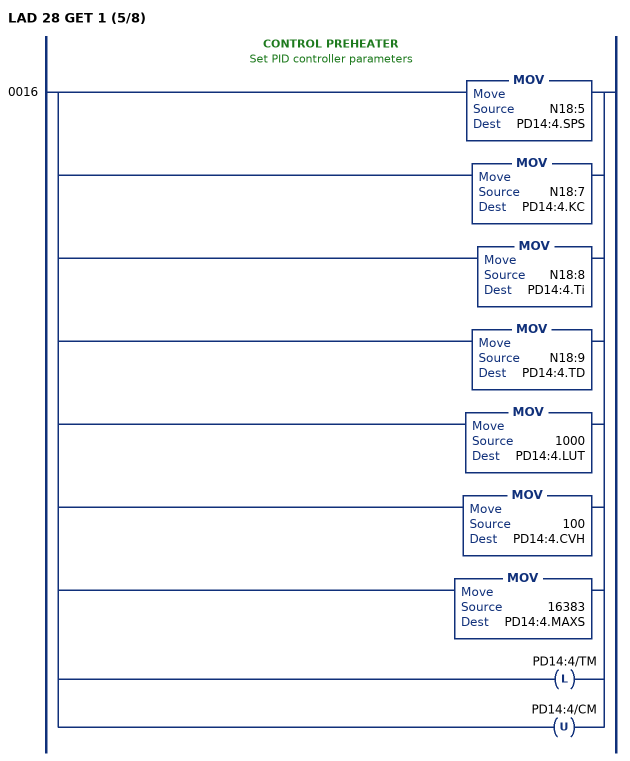
% Rung: 16 %
% TITLE: CONTROL PREHEATER %
% Set PID controller parameters %
SOR BST MOV N18:5 PD14:4.SPS NXB MOV N18:7 PD14:4.KC NXB MOV N18:8 PD14:4.Ti NXB MOV N18:9 PD14:4.TD NXB MOV 1000 PD14:4.LUT NXB MOV 100 PD14:4.CVH NXB MOV 16383 PD14:4.MAXS NXB OTL PD14:4/TM NXB OTU PD14:4/CM BND EOR
%   N18:5  GETTER_PH_SP  "<datalog>" %
%   N18:7  GET_PH_PID_GAIN %
%   N18:8  GET_PH_PID_INTEG %
%   N18:9  GET_PH_PID_DERIV %

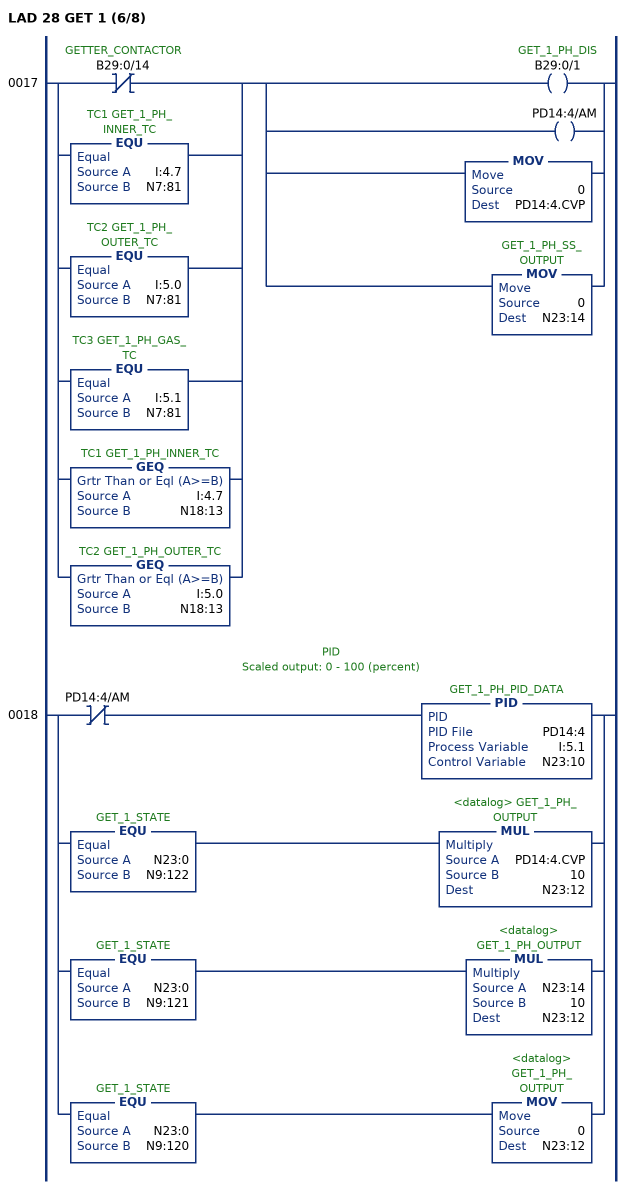
% Rung: 17 %
SOR BST XIO B29:0/14 NXB EQU I:4.7 N7:81 NXB EQU I:5.0 N7:81 NXB EQU I:5.1 N7:81 NXB GEQ I:4.7 N18:13 NXB GEQ I:5.0 N18:13 BND BST OTE B29:0/1 NXB OTE PD14:4/AM NXB MOV 0 PD14:4.CVP NXB MOV 0 N23:14 BND EOR
%   B29:0/14  GETTER_CONTACTOR %
%   I:4.7  GET_1_PH_INNER_TC  "TC1" %
%   N7:81  TC_OPEN_SP  "CONFIG The value read by an open TC input" %
%   I:5.0  GET_1_PH_OUTER_TC  "TC2" %
%   I:5.1  GET_1_PH_GAS_TC  "TC3" %
%   N18:13  GET_PH_ROD_LIMIT %
%   B29:0/1  GET_1_PH_DIS %
%   N23:14  GET_1_PH_SS_OUTPUT %
% Rung: 18 %
% PID
% Scaled output: 0 - 100 (percent) %
SOR BST XIO PD14:4/AM PID PD14:4 I:5.1 N23:10 NXB EQU N23:0 N9:122 MUL PD14:4.CVP 10 N23:12 NXB EQU N23:0 N9:121 MUL N23:14 10 N23:12 NXB EQU N23:0 N9:120 MOV 0 N23:12 BND EOR
%   PD14:4  GET_1_PH_PID_DATA %
%   I:5.1  GET_1_PH_GAS_TC  "TC3" %
%   N23:10  GET_1_PH_OUT_RAW %
%   N23:0  GET_1_STATE %
%   N9:122  GETTER_PURIFYING %
%   N23:12  GET_1_PH_OUTPUT  "<datalog>" %
%   N9:121  GETTER_SOFTSTART %
%   N23:14  GET_1_PH_SS_OUTPUT %
%   N9:120  GETTER_STANDBY %

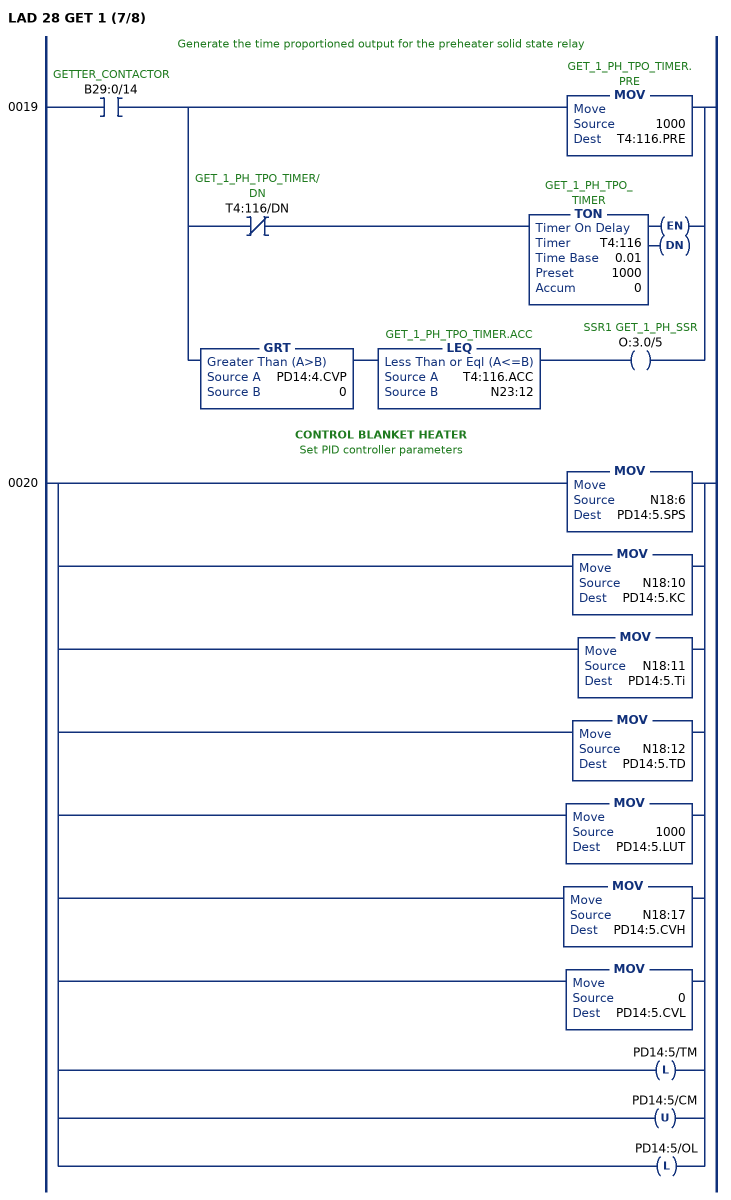
% Rung: 19 %
% Generate the time proportioned output for the preheater solid state relay %
SOR XIC B29:0/14 BST MOV 1000 T4:116.PRE NXB XIO T4:116/DN TON T4:116 0.01 1000 0 NXB GRT PD14:4.CVP 0 LEQ T4:116.ACC N23:12 OTE O:3.0/5 BND EOR
%   B29:0/14  GETTER_CONTACTOR %
%   T4:116  GET_1_PH_TPO_TIMER %
%   N23:12  GET_1_PH_OUTPUT  "<datalog>" %
%   O:3.0/5  GET_1_PH_SSR  "SSR1" %
% Rung: 20 %
% TITLE: CONTROL BLANKET HEATER %
% Set PID controller parameters %
SOR BST MOV N18:6 PD14:5.SPS NXB MOV N18:10 PD14:5.KC NXB MOV N18:11 PD14:5.Ti NXB MOV N18:12 PD14:5.TD NXB MOV 1000 PD14:5.LUT NXB MOV N18:17 PD14:5.CVH NXB MOV 0 PD14:5.CVL NXB OTL PD14:5/TM NXB OTU PD14:5/CM NXB OTL PD14:5/OL BND EOR
%   N18:6  GETTER_BLKT_SP  "<datalog>" %
%   N18:10  GET_BLKT_PID_GAIN %
%   N18:11  GET_BLKT_PID_INTEG %
%   N18:12  GET_BLKT_PID_DERIV %
%   N18:17  GET_BLKT_PID_HI_LIM %

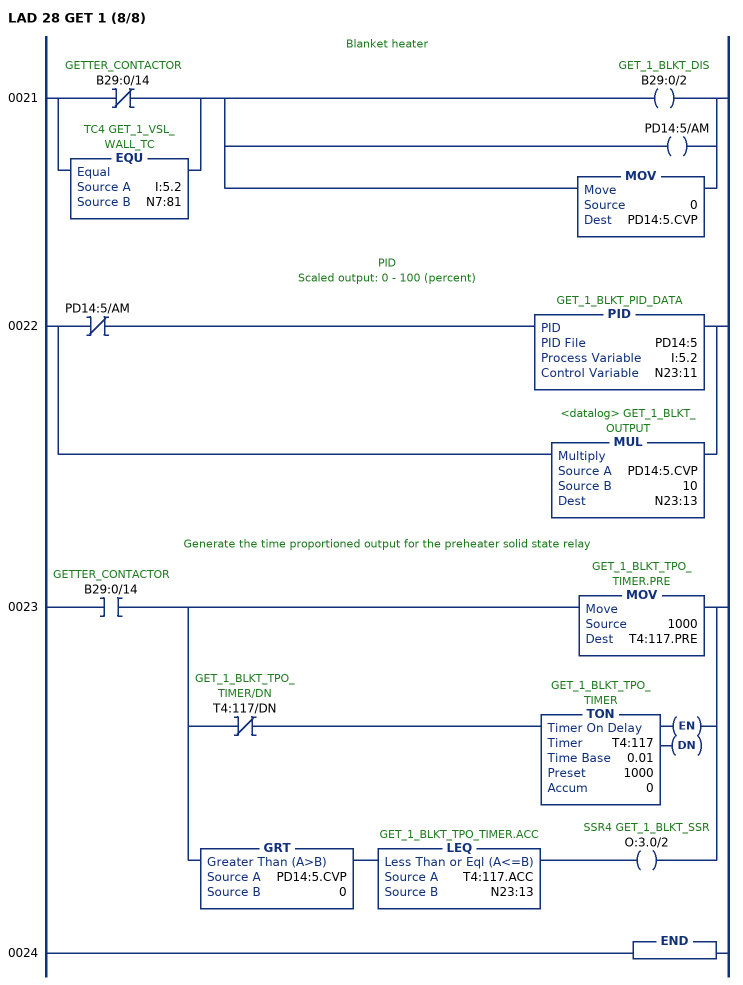
% Rung: 21 %
% Blanket heater %
SOR BST XIO B29:0/14 NXB EQU I:5.2 N7:81 BND BST OTE B29:0/2 NXB OTE PD14:5/AM NXB MOV 0 PD14:5.CVP BND EOR
%   B29:0/14  GETTER_CONTACTOR %
%   I:5.2  GET_1_VSL_WALL_TC  "TC4" %
%   N7:81  TC_OPEN_SP  "CONFIG The value read by an open TC input" %
%   B29:0/2  GET_1_BLKT_DIS %
% Rung: 22 %
% PID
% Scaled output: 0 - 100 (percent) %
SOR BST XIO PD14:5/AM PID PD14:5 I:5.2 N23:11 NXB MUL PD14:5.CVP 10 N23:13 BND EOR
%   PD14:5  GET_1_BLKT_PID_DATA %
%   I:5.2  GET_1_VSL_WALL_TC  "TC4" %
%   N23:11  GET_1_BLKT_OUT_RAW %
%   N23:13  GET_1_BLKT_OUTPUT  "<datalog>" %
% Rung: 23 %
% Generate the time proportioned output for the preheater solid state relay %
SOR XIC B29:0/14 BST MOV 1000 T4:117.PRE NXB XIO T4:117/DN TON T4:117 0.01 1000 0 NXB GRT PD14:5.CVP 0 LEQ T4:117.ACC N23:13 OTE O:3.0/2 BND EOR
%   B29:0/14  GETTER_CONTACTOR %
%   T4:117  GET_1_BLKT_TPO_TIMER %
%   N23:13  GET_1_BLKT_OUTPUT  "<datalog>" %
%   O:3.0/2  GET_1_BLKT_SSR  "SSR4" %
% Rung: 24 %
SOR END EOR

LADDER 29 "GET 2 FLT"
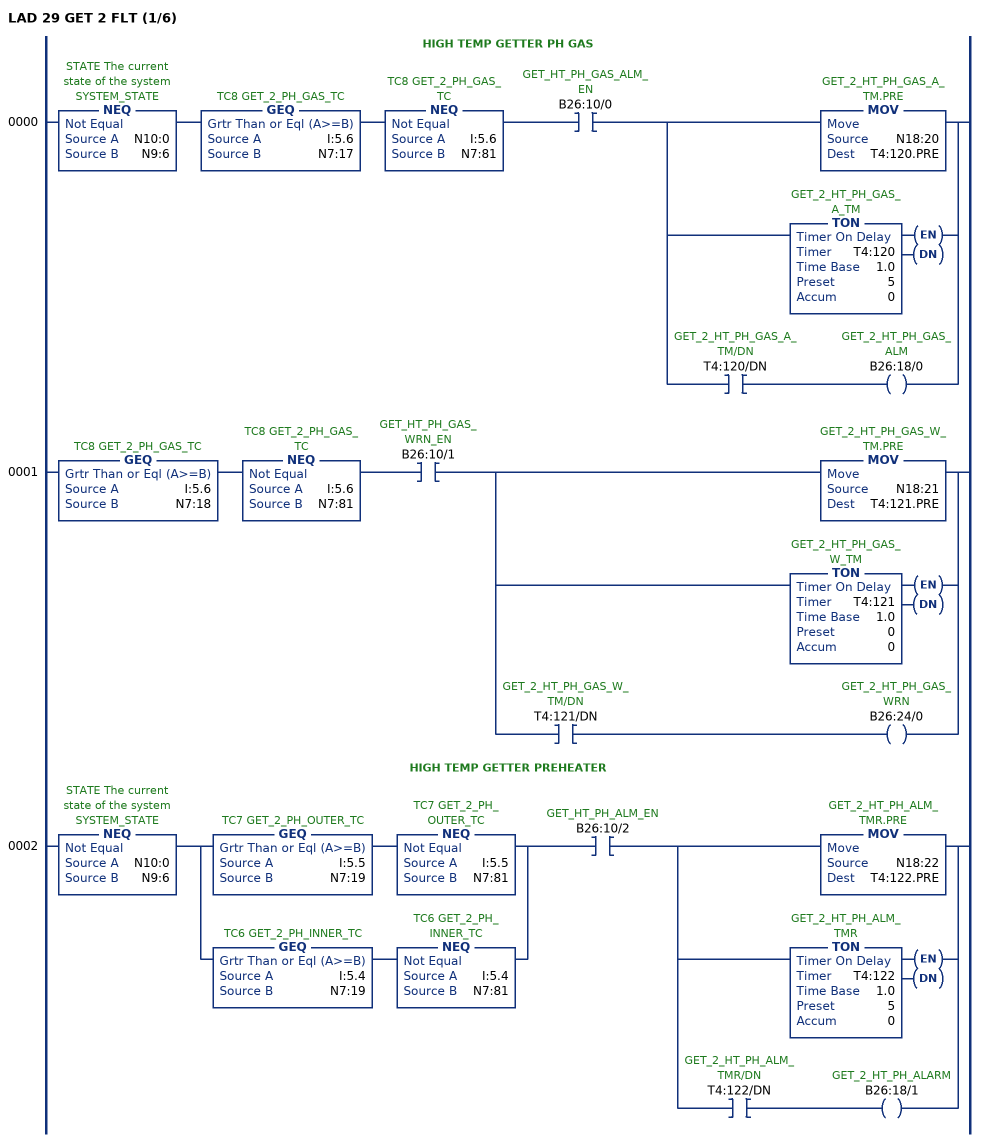
% Rung: 0 %
% TITLE: HIGH TEMP GETTER PH GAS %
SOR NEQ N10:0 N9:6 GEQ I:5.6 N7:17 NEQ I:5.6 N7:81 XIC B26:10/0 BST MOV N18:20 T4:120.PRE NXB TON T4:120 1.0 5 0 NXB XIC T4:120/DN OTE B26:18/0 BND EOR
%   N10:0  SYSTEM_STATE  "STATE The current state of the system" %
%   N9:6  SYSTEM_PURGE %
%   I:5.6  GET_2_PH_GAS_TC  "TC8" %
%   N7:17  GET_HT_PH_GAS_ALM_SP %
%   N7:81  TC_OPEN_SP  "CONFIG The value read by an open TC input" %
%   B26:10/0  GET_HT_PH_GAS_ALM_EN %
%   N18:20  GET_HT_PH_GAS_ALM_DL %
%   T4:120  GET_2_HT_PH_GAS_A_TM %
%   B26:18/0  GET_2_HT_PH_GAS_ALM %
% Rung: 1 %
SOR GEQ I:5.6 N7:18 NEQ I:5.6 N7:81 XIC B26:10/1 BST MOV N18:21 T4:121.PRE NXB TON T4:121 1.0 0 0 NXB XIC T4:121/DN OTE B26:24/0 BND EOR
%   I:5.6  GET_2_PH_GAS_TC  "TC8" %
%   N7:18  GET_HT_PH_GAS_WRN_SP %
%   N7:81  TC_OPEN_SP  "CONFIG The value read by an open TC input" %
%   B26:10/1  GET_HT_PH_GAS_WRN_EN %
%   N18:21  GET_HT_PH_GAS_WRN_DL %
%   T4:121  GET_2_HT_PH_GAS_W_TM %
%   B26:24/0  GET_2_HT_PH_GAS_WRN %
% Rung: 2 %
% TITLE: HIGH TEMP GETTER PREHEATER %
SOR NEQ N10:0 N9:6 BST GEQ I:5.5 N7:19 NEQ I:5.5 N7:81 NXB GEQ I:5.4 N7:19 NEQ I:5.4 N7:81 BND XIC B26:10/2 BST MOV N18:22 T4:122.PRE NXB TON T4:122 1.0 5 0 NXB XIC T4:122/DN OTE B26:18/1 BND EOR
%   N10:0  SYSTEM_STATE  "STATE The current state of the system" %
%   N9:6  SYSTEM_PURGE %
%   I:5.5  GET_2_PH_OUTER_TC  "TC7" %
%   N7:19  GET_HT_PH_ALM_SP %
%   N7:81  TC_OPEN_SP  "CONFIG The value read by an open TC input" %
%   I:5.4  GET_2_PH_INNER_TC  "TC6" %
%   B26:10/2  GET_HT_PH_ALM_EN %
%   N18:22  GET_HT_PH_ALM_DLY %
%   T4:122  GET_2_HT_PH_ALM_TMR %
%   B26:18/1  GET_2_HT_PH_ALARM %

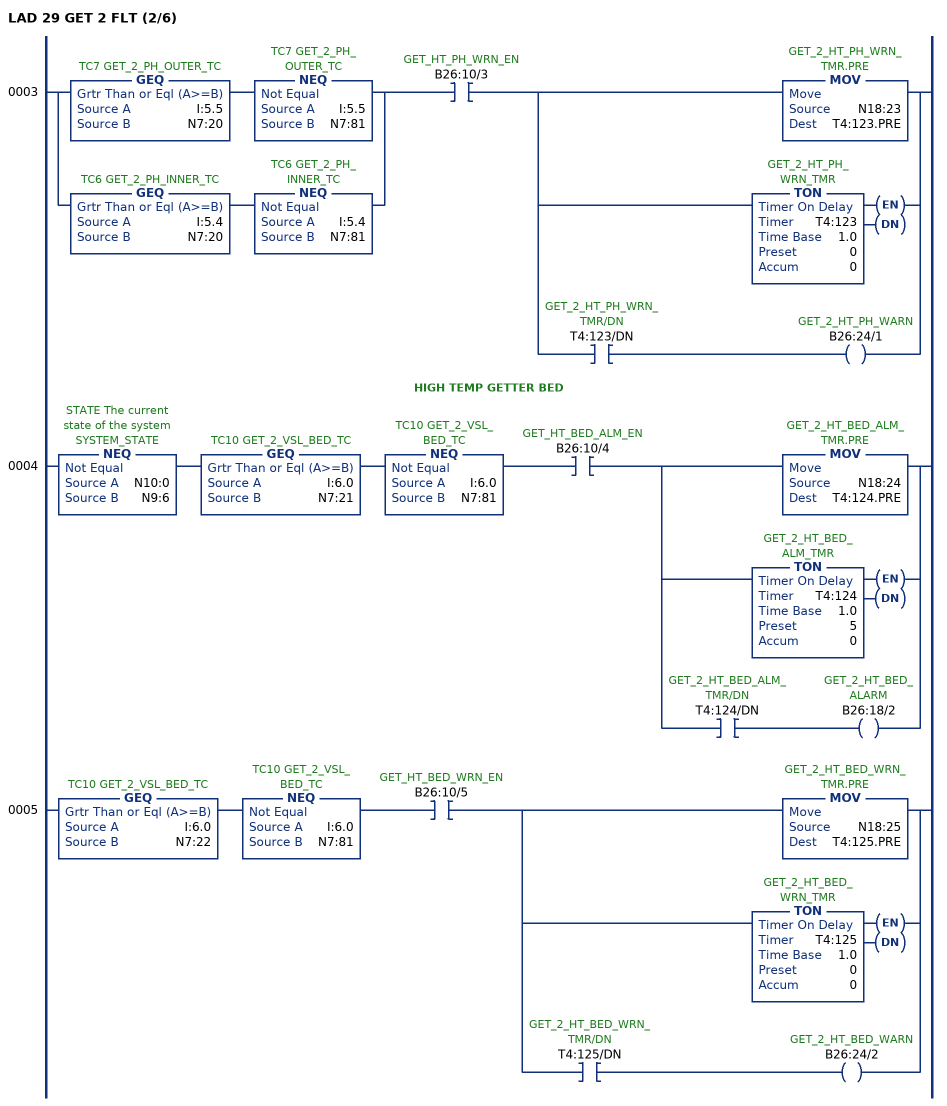
% Rung: 3 %
SOR BST GEQ I:5.5 N7:20 NEQ I:5.5 N7:81 NXB GEQ I:5.4 N7:20 NEQ I:5.4 N7:81 BND XIC B26:10/3 BST MOV N18:23 T4:123.PRE NXB TON T4:123 1.0 0 0 NXB XIC T4:123/DN OTE B26:24/1 BND EOR
%   I:5.5  GET_2_PH_OUTER_TC  "TC7" %
%   N7:20  GET_HT_PH_WRN_SP %
%   N7:81  TC_OPEN_SP  "CONFIG The value read by an open TC input" %
%   I:5.4  GET_2_PH_INNER_TC  "TC6" %
%   B26:10/3  GET_HT_PH_WRN_EN %
%   N18:23  GET_HT_PH_WRN_DLY %
%   T4:123  GET_2_HT_PH_WRN_TMR %
%   B26:24/1  GET_2_HT_PH_WARN %
% Rung: 4 %
% TITLE: HIGH TEMP GETTER BED %
SOR NEQ N10:0 N9:6 GEQ I:6.0 N7:21 NEQ I:6.0 N7:81 XIC B26:10/4 BST MOV N18:24 T4:124.PRE NXB TON T4:124 1.0 5 0 NXB XIC T4:124/DN OTE B26:18/2 BND EOR
%   N10:0  SYSTEM_STATE  "STATE The current state of the system" %
%   N9:6  SYSTEM_PURGE %
%   I:6.0  GET_2_VSL_BED_TC  "TC10" %
%   N7:21  GET_HT_BED_ALM_SP %
%   N7:81  TC_OPEN_SP  "CONFIG The value read by an open TC input" %
%   B26:10/4  GET_HT_BED_ALM_EN %
%   N18:24  GET_HT_BED_ALM_DLY %
%   T4:124  GET_2_HT_BED_ALM_TMR %
%   B26:18/2  GET_2_HT_BED_ALARM %
% Rung: 5 %
SOR GEQ I:6.0 N7:22 NEQ I:6.0 N7:81 XIC B26:10/5 BST MOV N18:25 T4:125.PRE NXB TON T4:125 1.0 0 0 NXB XIC T4:125/DN OTE B26:24/2 BND EOR
%   I:6.0  GET_2_VSL_BED_TC  "TC10" %
%   N7:22  GET_HT_BED_WRN_SP %
%   N7:81  TC_OPEN_SP  "CONFIG The value read by an open TC input" %
%   B26:10/5  GET_HT_BED_WRN_EN %
%   N18:25  GET_HT_BED_WRN_DLY %
%   T4:125  GET_2_HT_BED_WRN_TMR %
%   B26:24/2  GET_2_HT_BED_WARN %

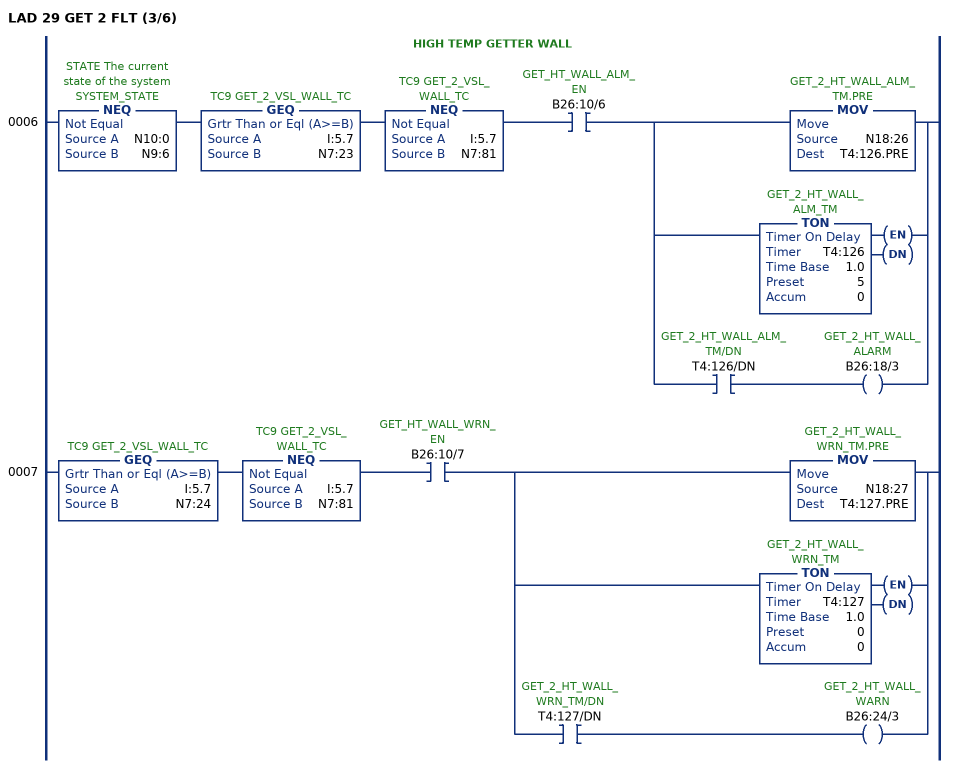
% Rung: 6 %
% TITLE: HIGH TEMP GETTER WALL %
SOR NEQ N10:0 N9:6 GEQ I:5.7 N7:23 NEQ I:5.7 N7:81 XIC B26:10/6 BST MOV N18:26 T4:126.PRE NXB TON T4:126 1.0 5 0 NXB XIC T4:126/DN OTE B26:18/3 BND EOR
%   N10:0  SYSTEM_STATE  "STATE The current state of the system" %
%   N9:6  SYSTEM_PURGE %
%   I:5.7  GET_2_VSL_WALL_TC  "TC9" %
%   N7:23  GET_HT_WALL_ALM_SP %
%   N7:81  TC_OPEN_SP  "CONFIG The value read by an open TC input" %
%   B26:10/6  GET_HT_WALL_ALM_EN %
%   N18:26  GET_HT_WALL_ALM_DLY %
%   T4:126  GET_2_HT_WALL_ALM_TM %
%   B26:18/3  GET_2_HT_WALL_ALARM %
% Rung: 7 %
SOR GEQ I:5.7 N7:24 NEQ I:5.7 N7:81 XIC B26:10/7 BST MOV N18:27 T4:127.PRE NXB TON T4:127 1.0 0 0 NXB XIC T4:127/DN OTE B26:24/3 BND EOR
%   I:5.7  GET_2_VSL_WALL_TC  "TC9" %
%   N7:24  GET_HT_WALL_WRN_SP %
%   N7:81  TC_OPEN_SP  "CONFIG The value read by an open TC input" %
%   B26:10/7  GET_HT_WALL_WRN_EN %
%   N18:27  GET_HT_WALL_WRN_DLY %
%   T4:127  GET_2_HT_WALL_WRN_TM %
%   B26:24/3  GET_2_HT_WALL_WARN %

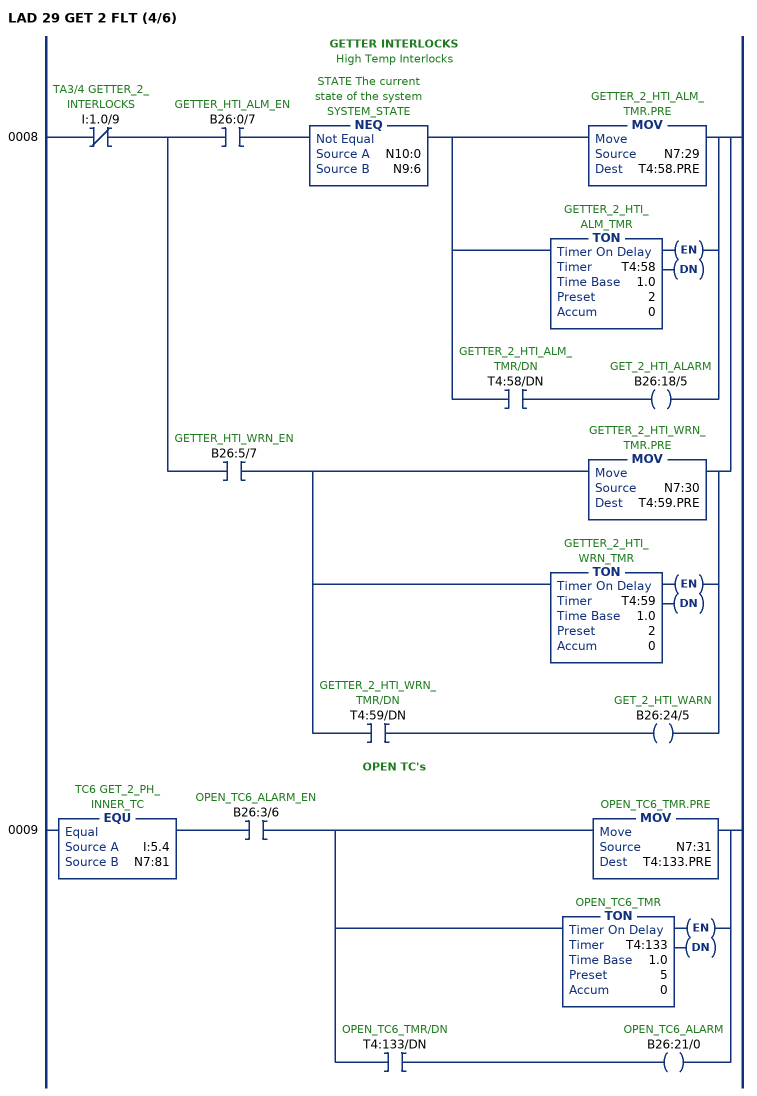
% Rung: 8 %
% TITLE: GETTER INTERLOCKS %
% High Temp Interlocks %
SOR XIO I:1.0/9 BST XIC B26:0/7 NEQ N10:0 N9:6 BST MOV N7:29 T4:58.PRE NXB TON T4:58 1.0 2 0 NXB XIC T4:58/DN OTE B26:18/5 BND NXB XIC B26:5/7 BST MOV N7:30 T4:59.PRE NXB TON T4:59 1.0 2 0 NXB XIC T4:59/DN OTE B26:24/5 BND BND EOR
%   I:1.0/9  GETTER_2_INTERLOCKS  "TA3/4" %
%   B26:0/7  GETTER_HTI_ALM_EN %
%   N10:0  SYSTEM_STATE  "STATE The current state of the system" %
%   N9:6  SYSTEM_PURGE %
%   N7:29  GETTER_HTI_ALM_DLY %
%   T4:58  GETTER_2_HTI_ALM_TMR %
%   B26:18/5  GET_2_HTI_ALARM %
%   B26:5/7  GETTER_HTI_WRN_EN %
%   N7:30  GETTER_HTI_WRN_DLY %
%   T4:59  GETTER_2_HTI_WRN_TMR %
%   B26:24/5  GET_2_HTI_WARN %
% Rung: 9 %
% TITLE: OPEN TC's %
SOR EQU I:5.4 N7:81 XIC B26:3/6 BST MOV N7:31 T4:133.PRE NXB TON T4:133 1.0 5 0 NXB XIC T4:133/DN OTE B26:21/0 BND EOR
%   I:5.4  GET_2_PH_INNER_TC  "TC6" %
%   N7:81  TC_OPEN_SP  "CONFIG The value read by an open TC input" %
%   B26:3/6  OPEN_TC6_ALARM_EN %
%   N7:31  OPEN_TC_DLY %
%   T4:133  OPEN_TC6_TMR %
%   B26:21/0  OPEN_TC6_ALARM %

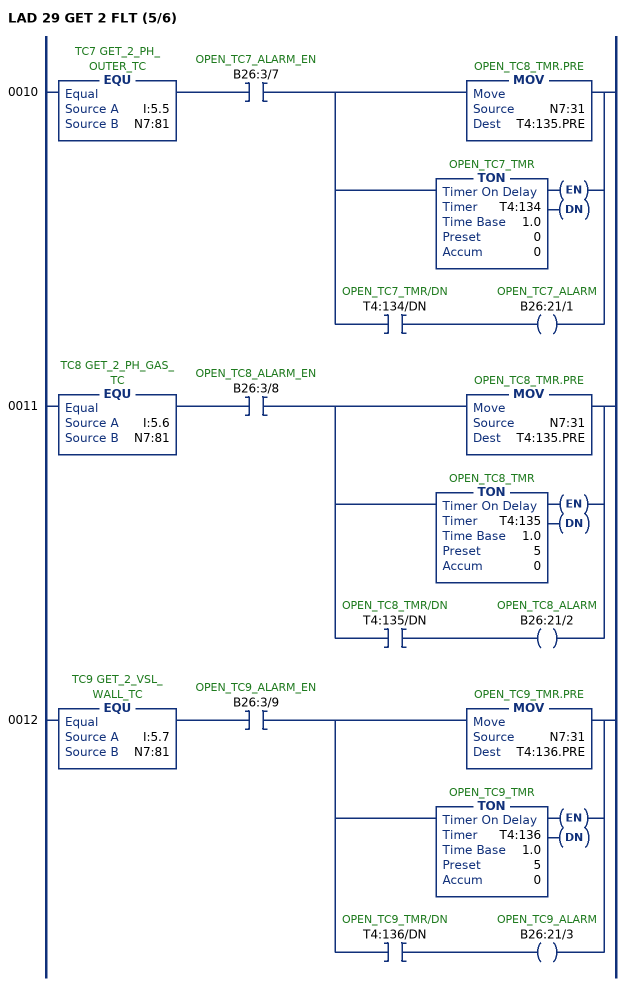
% Rung: 10 %
SOR EQU I:5.5 N7:81 XIC B26:3/7 BST MOV N7:31 T4:135.PRE NXB TON T4:134 1.0 0 0 NXB XIC T4:134/DN OTE B26:21/1 BND EOR
%   I:5.5  GET_2_PH_OUTER_TC  "TC7" %
%   N7:81  TC_OPEN_SP  "CONFIG The value read by an open TC input" %
%   B26:3/7  OPEN_TC7_ALARM_EN %
%   N7:31  OPEN_TC_DLY %
%   T4:135  OPEN_TC8_TMR %
%   T4:134  OPEN_TC7_TMR %
%   B26:21/1  OPEN_TC7_ALARM %
% Rung: 11 %
SOR EQU I:5.6 N7:81 XIC B26:3/8 BST MOV N7:31 T4:135.PRE NXB TON T4:135 1.0 5 0 NXB XIC T4:135/DN OTE B26:21/2 BND EOR
%   I:5.6  GET_2_PH_GAS_TC  "TC8" %
%   N7:81  TC_OPEN_SP  "CONFIG The value read by an open TC input" %
%   B26:3/8  OPEN_TC8_ALARM_EN %
%   N7:31  OPEN_TC_DLY %
%   T4:135  OPEN_TC8_TMR %
%   B26:21/2  OPEN_TC8_ALARM %
% Rung: 12 %
SOR EQU I:5.7 N7:81 XIC B26:3/9 BST MOV N7:31 T4:136.PRE NXB TON T4:136 1.0 5 0 NXB XIC T4:136/DN OTE B26:21/3 BND EOR
%   I:5.7  GET_2_VSL_WALL_TC  "TC9" %
%   N7:81  TC_OPEN_SP  "CONFIG The value read by an open TC input" %
%   B26:3/9  OPEN_TC9_ALARM_EN %
%   N7:31  OPEN_TC_DLY %
%   T4:136  OPEN_TC9_TMR %
%   B26:21/3  OPEN_TC9_ALARM %

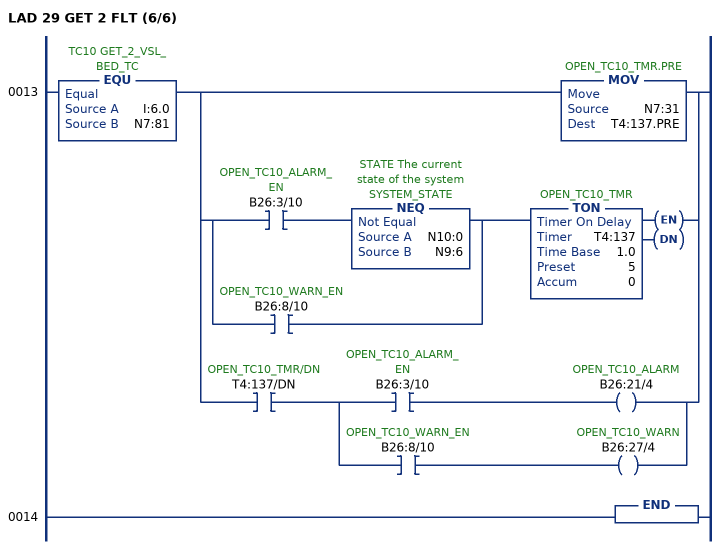
% Rung: 13 %
SOR EQU I:6.0 N7:81 BST MOV N7:31 T4:137.PRE NXB BST XIC B26:3/10 NEQ N10:0 N9:6 NXB XIC B26:8/10 BND TON T4:137 1.0 5 0 NXB XIC T4:137/DN BST XIC B26:3/10 OTE B26:21/4 NXB XIC B26:8/10 OTE B26:27/4 BND BND EOR
%   I:6.0  GET_2_VSL_BED_TC  "TC10" %
%   N7:81  TC_OPEN_SP  "CONFIG The value read by an open TC input" %
%   N7:31  OPEN_TC_DLY %
%   T4:137  OPEN_TC10_TMR %
%   B26:3/10  OPEN_TC10_ALARM_EN %
%   N10:0  SYSTEM_STATE  "STATE The current state of the system" %
%   N9:6  SYSTEM_PURGE %
%   B26:8/10  OPEN_TC10_WARN_EN %
%   B26:21/4  OPEN_TC10_ALARM %
%   B26:27/4  OPEN_TC10_WARN %
% Rung: 14 %
SOR END EOR

LADDER 30 "GET 2"
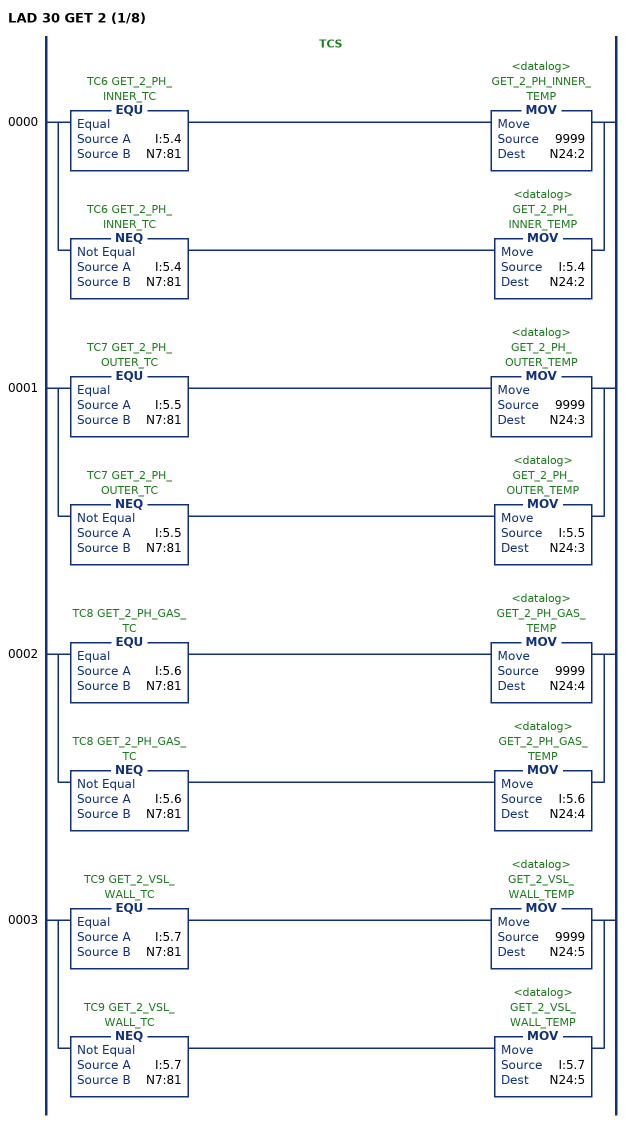
% Rung: 0 %
% TITLE: TCS %
SOR BST EQU I:5.4 N7:81 MOV 9999 N24:2 NXB NEQ I:5.4 N7:81 MOV I:5.4 N24:2 BND EOR
%   I:5.4  GET_2_PH_INNER_TC  "TC6" %
%   N7:81  TC_OPEN_SP  "CONFIG The value read by an open TC input" %
%   N24:2  GET_2_PH_INNER_TEMP  "<datalog>" %
% Rung: 1 %
SOR BST EQU I:5.5 N7:81 MOV 9999 N24:3 NXB NEQ I:5.5 N7:81 MOV I:5.5 N24:3 BND EOR
%   I:5.5  GET_2_PH_OUTER_TC  "TC7" %
%   N7:81  TC_OPEN_SP  "CONFIG The value read by an open TC input" %
%   N24:3  GET_2_PH_OUTER_TEMP  "<datalog>" %
% Rung: 2 %
SOR BST EQU I:5.6 N7:81 MOV 9999 N24:4 NXB NEQ I:5.6 N7:81 MOV I:5.6 N24:4 BND EOR
%   I:5.6  GET_2_PH_GAS_TC  "TC8" %
%   N7:81  TC_OPEN_SP  "CONFIG The value read by an open TC input" %
%   N24:4  GET_2_PH_GAS_TEMP  "<datalog>" %
% Rung: 3 %
SOR BST EQU I:5.7 N7:81 MOV 9999 N24:5 NXB NEQ I:5.7 N7:81 MOV I:5.7 N24:5 BND EOR
%   I:5.7  GET_2_VSL_WALL_TC  "TC9" %
%   N7:81  TC_OPEN_SP  "CONFIG The value read by an open TC input" %
%   N24:5  GET_2_VSL_WALL_TEMP  "<datalog>" %

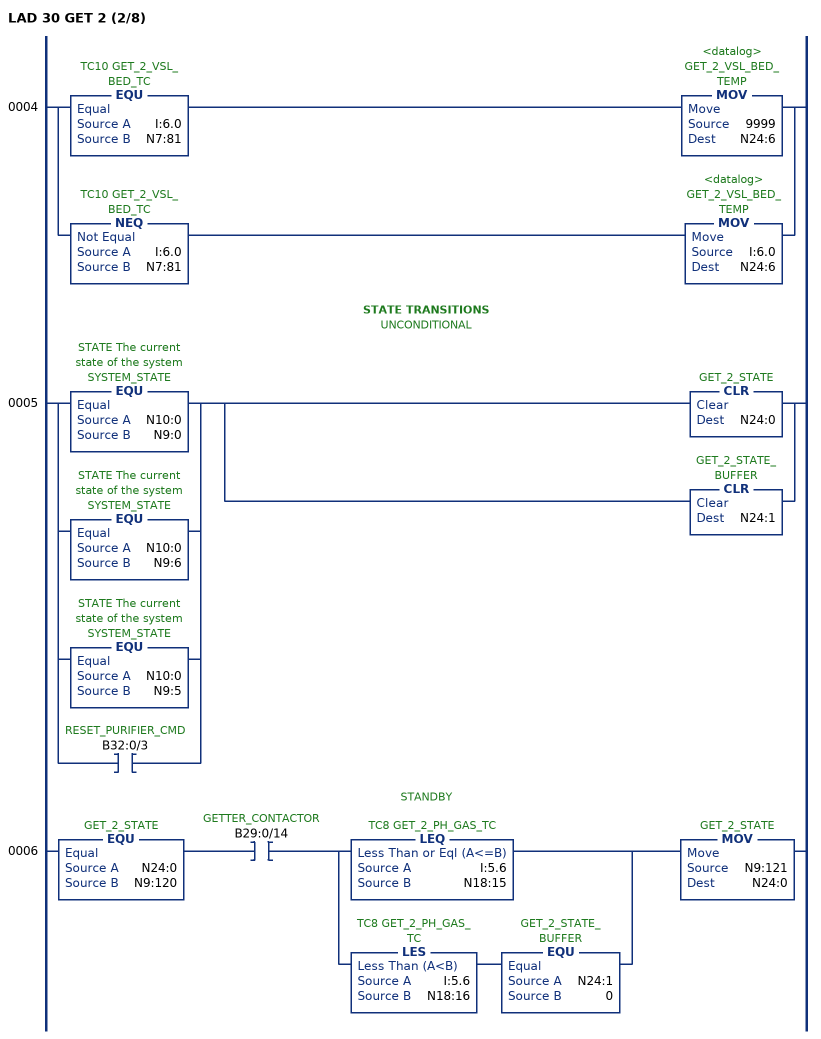
% Rung: 4 %
SOR BST EQU I:6.0 N7:81 MOV 9999 N24:6 NXB NEQ I:6.0 N7:81 MOV I:6.0 N24:6 BND EOR
%   I:6.0  GET_2_VSL_BED_TC  "TC10" %
%   N7:81  TC_OPEN_SP  "CONFIG The value read by an open TC input" %
%   N24:6  GET_2_VSL_BED_TEMP  "<datalog>" %
% Rung: 5 %
% TITLE: STATE TRANSITIONS %
% UNCONDITIONAL %
SOR BST EQU N10:0 N9:0 NXB EQU N10:0 N9:6 NXB EQU N10:0 N9:5 NXB XIC B32:0/3 BND BST CLR N24:0 NXB CLR N24:1 BND EOR
%   N10:0  SYSTEM_STATE  "STATE The current state of the system" %
%   N9:0  SYSTEM_OFFLINE %
%   N9:6  SYSTEM_PURGE %
%   N9:5  SYSTEM_QUICK_START %
%   B32:0/3  RESET_PURIFIER_CMD %
%   N24:0  GET_2_STATE %
%   N24:1  GET_2_STATE_BUFFER %
% Rung: 6 %
% STANDBY %
SOR EQU N24:0 N9:120 XIC B29:0/14 BST LEQ I:5.6 N18:15 NXB LES I:5.6 N18:16 EQU N24:1 0 BND MOV N9:121 N24:0 EOR
%   N24:0  GET_2_STATE %
%   N9:120  GETTER_STANDBY %
%   B29:0/14  GETTER_CONTACTOR %
%   I:5.6  GET_2_PH_GAS_TC  "TC8" %
%   N18:15  GETTER_SS_BEGIN_TEMP %
%   N18:16  GETTER_SS_END_TEMP %
%   N24:1  GET_2_STATE_BUFFER %
%   N9:121  GETTER_SOFTSTART %

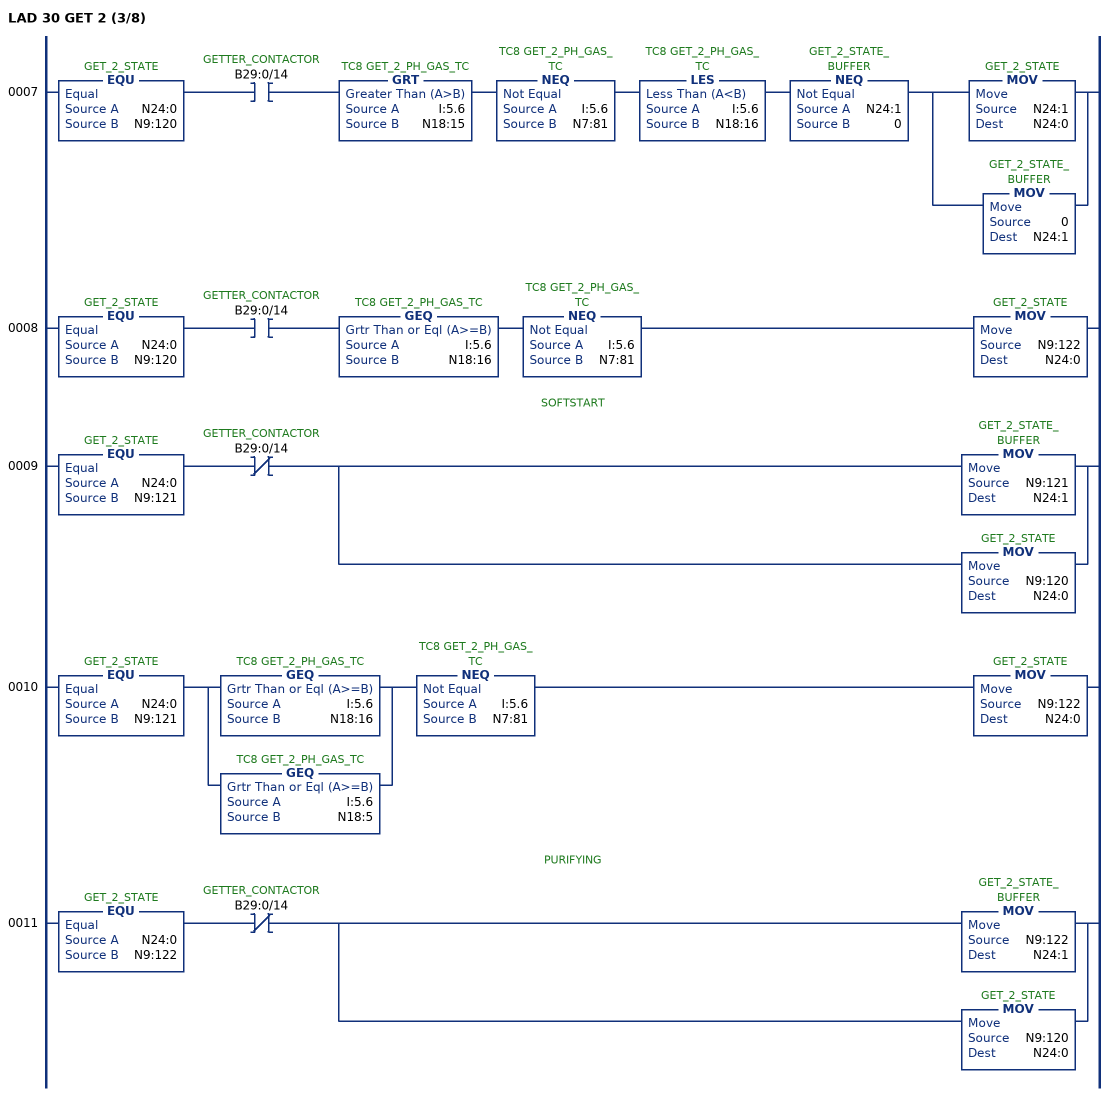
% Rung: 7 %
SOR EQU N24:0 N9:120 XIC B29:0/14 GRT I:5.6 N18:15 NEQ I:5.6 N7:81 LES I:5.6 N18:16 NEQ N24:1 0 BST MOV N24:1 N24:0 NXB MOV 0 N24:1 BND EOR
%   N24:0  GET_2_STATE %
%   N9:120  GETTER_STANDBY %
%   B29:0/14  GETTER_CONTACTOR %
%   I:5.6  GET_2_PH_GAS_TC  "TC8" %
%   N18:15  GETTER_SS_BEGIN_TEMP %
%   N7:81  TC_OPEN_SP  "CONFIG The value read by an open TC input" %
%   N18:16  GETTER_SS_END_TEMP %
%   N24:1  GET_2_STATE_BUFFER %
% Rung: 8 %
SOR EQU N24:0 N9:120 XIC B29:0/14 GEQ I:5.6 N18:16 NEQ I:5.6 N7:81 MOV N9:122 N24:0 EOR
%   N24:0  GET_2_STATE %
%   N9:120  GETTER_STANDBY %
%   B29:0/14  GETTER_CONTACTOR %
%   I:5.6  GET_2_PH_GAS_TC  "TC8" %
%   N18:16  GETTER_SS_END_TEMP %
%   N7:81  TC_OPEN_SP  "CONFIG The value read by an open TC input" %
%   N9:122  GETTER_PURIFYING %
% Rung: 9 %
% SOFTSTART %
SOR EQU N24:0 N9:121 XIO B29:0/14 BST MOV N9:121 N24:1 NXB MOV N9:120 N24:0 BND EOR
%   N24:0  GET_2_STATE %
%   N9:121  GETTER_SOFTSTART %
%   B29:0/14  GETTER_CONTACTOR %
%   N24:1  GET_2_STATE_BUFFER %
%   N9:120  GETTER_STANDBY %
% Rung: 10 %
SOR EQU N24:0 N9:121 BST GEQ I:5.6 N18:16 NXB GEQ I:5.6 N18:5 BND NEQ I:5.6 N7:81 MOV N9:122 N24:0 EOR
%   N24:0  GET_2_STATE %
%   N9:121  GETTER_SOFTSTART %
%   I:5.6  GET_2_PH_GAS_TC  "TC8" %
%   N18:16  GETTER_SS_END_TEMP %
%   N18:5  GETTER_PH_SP  "<datalog>" %
%   N7:81  TC_OPEN_SP  "CONFIG The value read by an open TC input" %
%   N9:122  GETTER_PURIFYING %
% Rung: 11 %
% PURIFYING %
SOR EQU N24:0 N9:122 XIO B29:0/14 BST MOV N9:122 N24:1 NXB MOV N9:120 N24:0 BND EOR
%   N24:0  GET_2_STATE %
%   N9:122  GETTER_PURIFYING %
%   B29:0/14  GETTER_CONTACTOR %
%   N24:1  GET_2_STATE_BUFFER %
%   N9:120  GETTER_STANDBY %

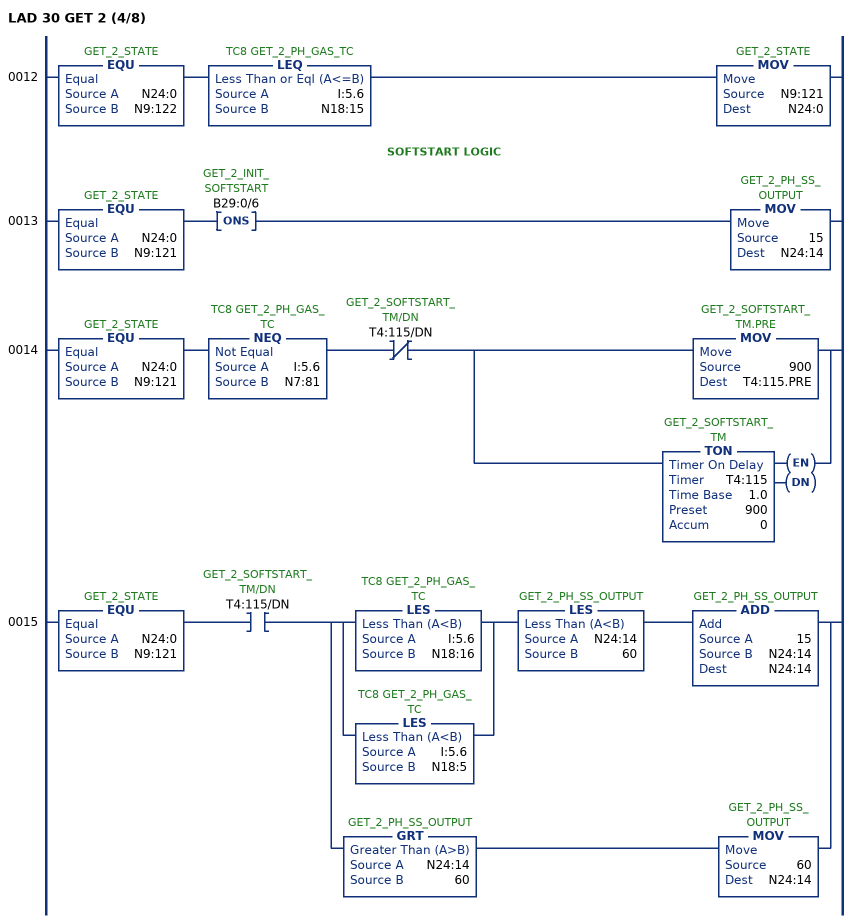
% Rung: 12 %
SOR EQU N24:0 N9:122 LEQ I:5.6 N18:15 MOV N9:121 N24:0 EOR
%   N24:0  GET_2_STATE %
%   N9:122  GETTER_PURIFYING %
%   I:5.6  GET_2_PH_GAS_TC  "TC8" %
%   N18:15  GETTER_SS_BEGIN_TEMP %
%   N9:121  GETTER_SOFTSTART %
% Rung: 13 %
% TITLE: SOFTSTART LOGIC %
SOR EQU N24:0 N9:121 ONS B29:0/6 MOV 15 N24:14 EOR
%   N24:0  GET_2_STATE %
%   N9:121  GETTER_SOFTSTART %
%   B29:0/6  GET_2_INIT_SOFTSTART %
%   N24:14  GET_2_PH_SS_OUTPUT %
% Rung: 14 %
SOR EQU N24:0 N9:121 NEQ I:5.6 N7:81 XIO T4:115/DN BST MOV 900 T4:115.PRE NXB TON T4:115 1.0 900 0 BND EOR
%   N24:0  GET_2_STATE %
%   N9:121  GETTER_SOFTSTART %
%   I:5.6  GET_2_PH_GAS_TC  "TC8" %
%   N7:81  TC_OPEN_SP  "CONFIG The value read by an open TC input" %
%   T4:115  GET_2_SOFTSTART_TM %
% Rung: 15 %
SOR EQU N24:0 N9:121 XIC T4:115/DN BST BST LES I:5.6 N18:16 NXB LES I:5.6 N18:5 BND LES N24:14 60 ADD 15 N24:14 N24:14 NXB GRT N24:14 60 MOV 60 N24:14 BND EOR
%   N24:0  GET_2_STATE %
%   N9:121  GETTER_SOFTSTART %
%   T4:115  GET_2_SOFTSTART_TM %
%   I:5.6  GET_2_PH_GAS_TC  "TC8" %
%   N18:16  GETTER_SS_END_TEMP %
%   N18:5  GETTER_PH_SP  "<datalog>" %
%   N24:14  GET_2_PH_SS_OUTPUT %

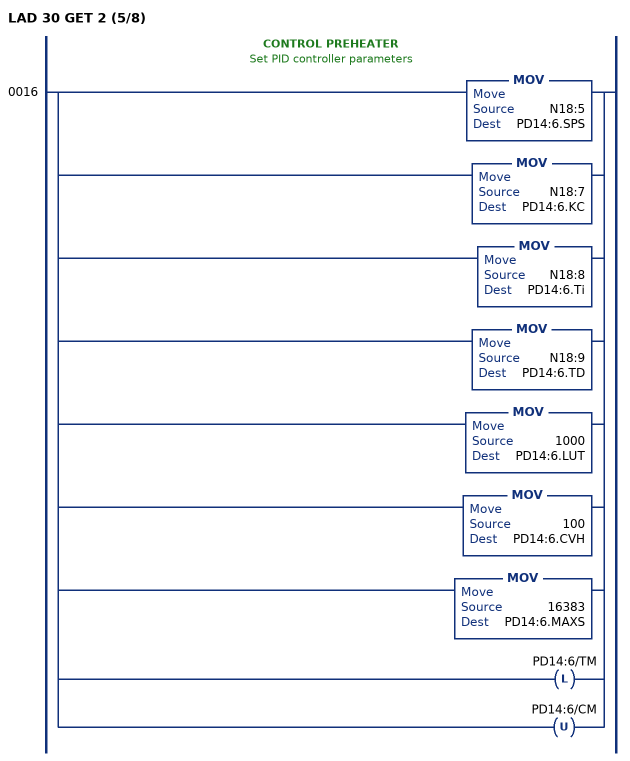
% Rung: 16 %
% TITLE: CONTROL PREHEATER %
% Set PID controller parameters %
SOR BST MOV N18:5 PD14:6.SPS NXB MOV N18:7 PD14:6.KC NXB MOV N18:8 PD14:6.Ti NXB MOV N18:9 PD14:6.TD NXB MOV 1000 PD14:6.LUT NXB MOV 100 PD14:6.CVH NXB MOV 16383 PD14:6.MAXS NXB OTL PD14:6/TM NXB OTU PD14:6/CM BND EOR
%   N18:5  GETTER_PH_SP  "<datalog>" %
%   N18:7  GET_PH_PID_GAIN %
%   N18:8  GET_PH_PID_INTEG %
%   N18:9  GET_PH_PID_DERIV %

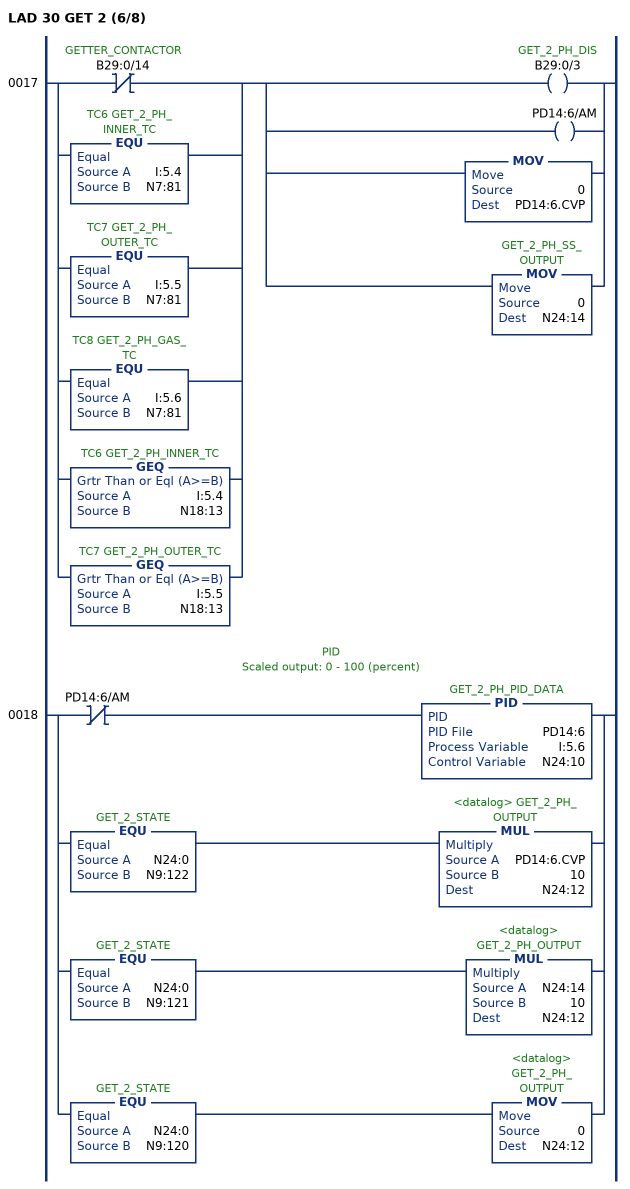
% Rung: 17 %
SOR BST XIO B29:0/14 NXB EQU I:5.4 N7:81 NXB EQU I:5.5 N7:81 NXB EQU I:5.6 N7:81 NXB GEQ I:5.4 N18:13 NXB GEQ I:5.5 N18:13 BND BST OTE B29:0/3 NXB OTE PD14:6/AM NXB MOV 0 PD14:6.CVP NXB MOV 0 N24:14 BND EOR
%   B29:0/14  GETTER_CONTACTOR %
%   I:5.4  GET_2_PH_INNER_TC  "TC6" %
%   N7:81  TC_OPEN_SP  "CONFIG The value read by an open TC input" %
%   I:5.5  GET_2_PH_OUTER_TC  "TC7" %
%   I:5.6  GET_2_PH_GAS_TC  "TC8" %
%   N18:13  GET_PH_ROD_LIMIT %
%   B29:0/3  GET_2_PH_DIS %
%   N24:14  GET_2_PH_SS_OUTPUT %
% Rung: 18 %
% PID
% Scaled output: 0 - 100 (percent) %
SOR BST XIO PD14:6/AM PID PD14:6 I:5.6 N24:10 NXB EQU N24:0 N9:122 MUL PD14:6.CVP 10 N24:12 NXB EQU N24:0 N9:121 MUL N24:14 10 N24:12 NXB EQU N24:0 N9:120 MOV 0 N24:12 BND EOR
%   PD14:6  GET_2_PH_PID_DATA %
%   I:5.6  GET_2_PH_GAS_TC  "TC8" %
%   N24:10  GET_2_PH_OUT_RAW %
%   N24:0  GET_2_STATE %
%   N9:122  GETTER_PURIFYING %
%   N24:12  GET_2_PH_OUTPUT  "<datalog>" %
%   N9:121  GETTER_SOFTSTART %
%   N24:14  GET_2_PH_SS_OUTPUT %
%   N9:120  GETTER_STANDBY %

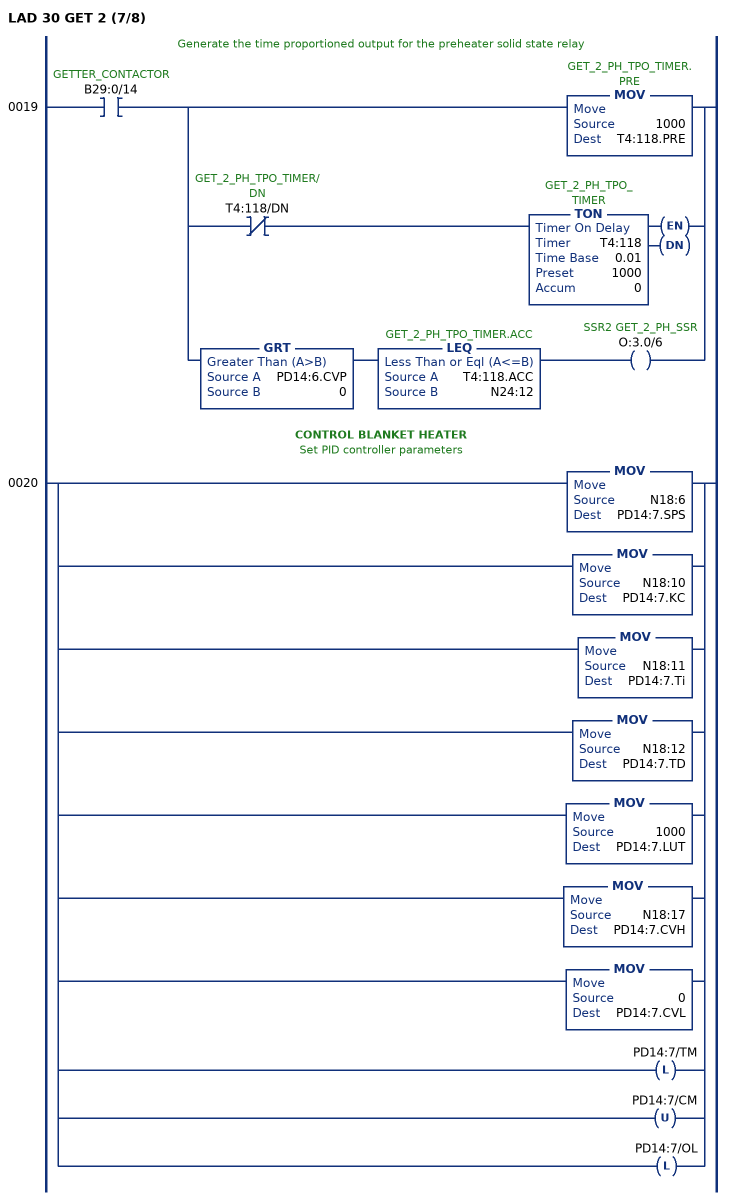
% Rung: 19 %
% Generate the time proportioned output for the preheater solid state relay %
SOR XIC B29:0/14 BST MOV 1000 T4:118.PRE NXB XIO T4:118/DN TON T4:118 0.01 1000 0 NXB GRT PD14:6.CVP 0 LEQ T4:118.ACC N24:12 OTE O:3.0/6 BND EOR
%   B29:0/14  GETTER_CONTACTOR %
%   T4:118  GET_2_PH_TPO_TIMER %
%   N24:12  GET_2_PH_OUTPUT  "<datalog>" %
%   O:3.0/6  GET_2_PH_SSR  "SSR2" %
% Rung: 20 %
% TITLE: CONTROL BLANKET HEATER %
% Set PID controller parameters %
SOR BST MOV N18:6 PD14:7.SPS NXB MOV N18:10 PD14:7.KC NXB MOV N18:11 PD14:7.Ti NXB MOV N18:12 PD14:7.TD NXB MOV 1000 PD14:7.LUT NXB MOV N18:17 PD14:7.CVH NXB MOV 0 PD14:7.CVL NXB OTL PD14:7/TM NXB OTU PD14:7/CM NXB OTL PD14:7/OL BND EOR
%   N18:6  GETTER_BLKT_SP  "<datalog>" %
%   N18:10  GET_BLKT_PID_GAIN %
%   N18:11  GET_BLKT_PID_INTEG %
%   N18:12  GET_BLKT_PID_DERIV %
%   N18:17  GET_BLKT_PID_HI_LIM %

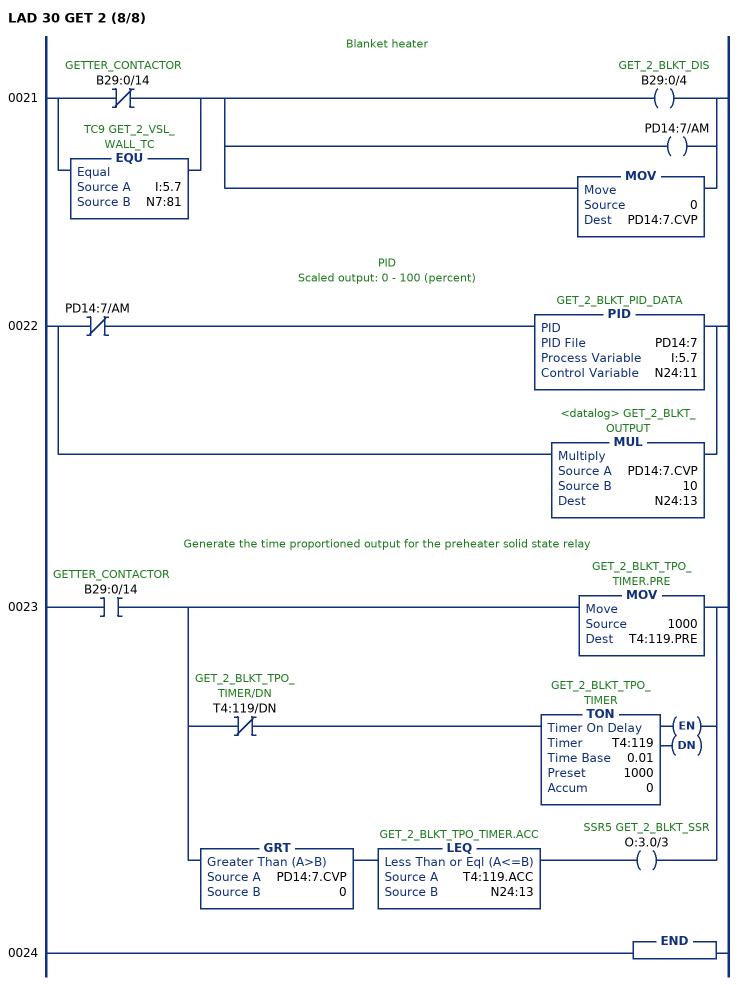
% Rung: 21 %
% Blanket heater %
SOR BST XIO B29:0/14 NXB EQU I:5.7 N7:81 BND BST OTE B29:0/4 NXB OTE PD14:7/AM NXB MOV 0 PD14:7.CVP BND EOR
%   B29:0/14  GETTER_CONTACTOR %
%   I:5.7  GET_2_VSL_WALL_TC  "TC9" %
%   N7:81  TC_OPEN_SP  "CONFIG The value read by an open TC input" %
%   B29:0/4  GET_2_BLKT_DIS %
% Rung: 22 %
% PID
% Scaled output: 0 - 100 (percent) %
SOR BST XIO PD14:7/AM PID PD14:7 I:5.7 N24:11 NXB MUL PD14:7.CVP 10 N24:13 BND EOR
%   PD14:7  GET_2_BLKT_PID_DATA %
%   I:5.7  GET_2_VSL_WALL_TC  "TC9" %
%   N24:11  GET_2_BLKT_OUT_RAW %
%   N24:13  GET_2_BLKT_OUTPUT  "<datalog>" %
% Rung: 23 %
% Generate the time proportioned output for the preheater solid state relay %
SOR XIC B29:0/14 BST MOV 1000 T4:119.PRE NXB XIO T4:119/DN TON T4:119 0.01 1000 0 NXB GRT PD14:7.CVP 0 LEQ T4:119.ACC N24:13 OTE O:3.0/3 BND EOR
%   B29:0/14  GETTER_CONTACTOR %
%   T4:119  GET_2_BLKT_TPO_TIMER %
%   N24:13  GET_2_BLKT_OUTPUT  "<datalog>" %
%   O:3.0/3  GET_2_BLKT_SSR  "SSR5" %
% Rung: 24 %
SOR END EOR

LADDER 31 "GET 3 FLT"
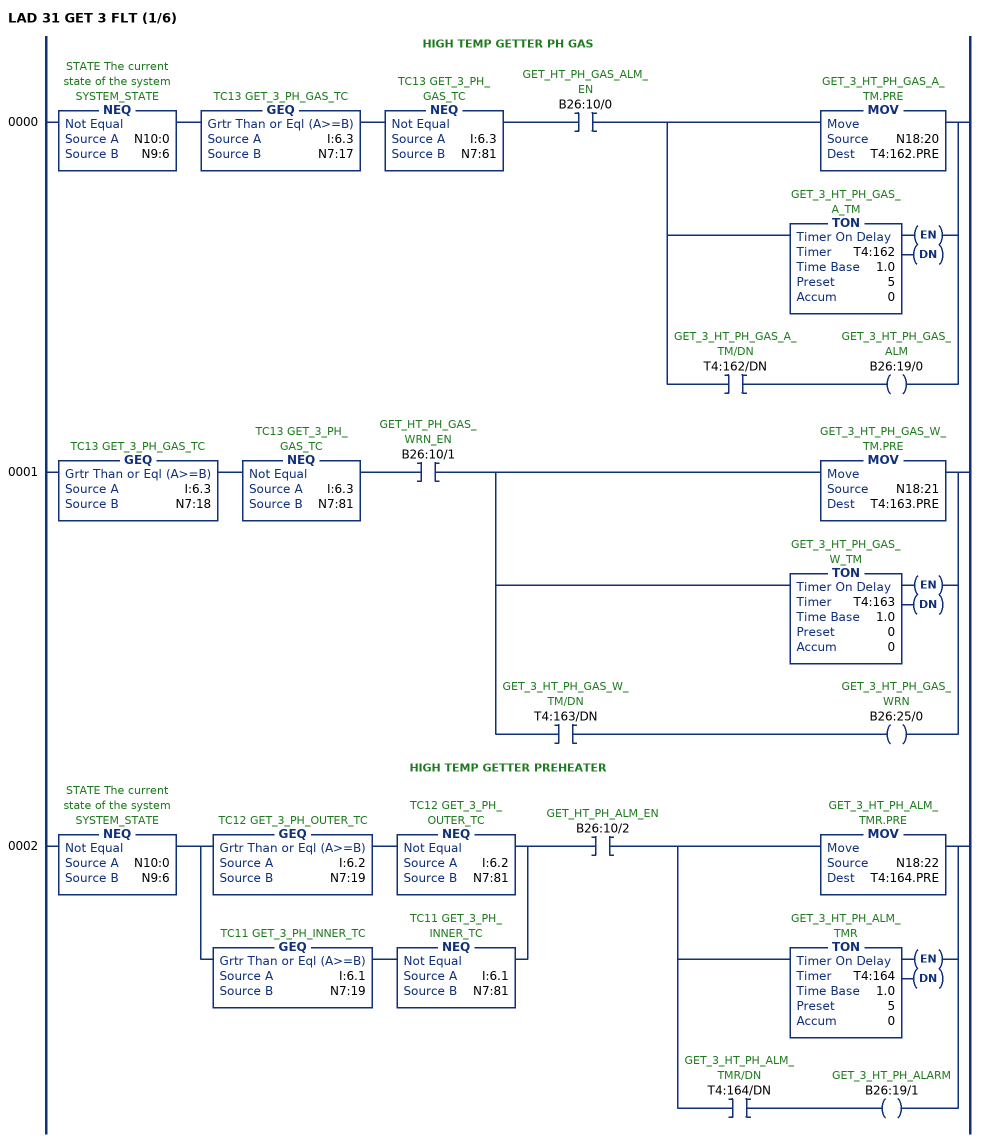
% Rung: 0 %
% TITLE: HIGH TEMP GETTER PH GAS %
SOR NEQ N10:0 N9:6 GEQ I:6.3 N7:17 NEQ I:6.3 N7:81 XIC B26:10/0 BST MOV N18:20 T4:162.PRE NXB TON T4:162 1.0 5 0 NXB XIC T4:162/DN OTE B26:19/0 BND EOR
%   N10:0  SYSTEM_STATE  "STATE The current state of the system" %
%   N9:6  SYSTEM_PURGE %
%   I:6.3  GET_3_PH_GAS_TC  "TC13" %
%   N7:17  GET_HT_PH_GAS_ALM_SP %
%   N7:81  TC_OPEN_SP  "CONFIG The value read by an open TC input" %
%   B26:10/0  GET_HT_PH_GAS_ALM_EN %
%   N18:20  GET_HT_PH_GAS_ALM_DL %
%   T4:162  GET_3_HT_PH_GAS_A_TM %
%   B26:19/0  GET_3_HT_PH_GAS_ALM %
% Rung: 1 %
SOR GEQ I:6.3 N7:18 NEQ I:6.3 N7:81 XIC B26:10/1 BST MOV N18:21 T4:163.PRE NXB TON T4:163 1.0 0 0 NXB XIC T4:163/DN OTE B26:25/0 BND EOR
%   I:6.3  GET_3_PH_GAS_TC  "TC13" %
%   N7:18  GET_HT_PH_GAS_WRN_SP %
%   N7:81  TC_OPEN_SP  "CONFIG The value read by an open TC input" %
%   B26:10/1  GET_HT_PH_GAS_WRN_EN %
%   N18:21  GET_HT_PH_GAS_WRN_DL %
%   T4:163  GET_3_HT_PH_GAS_W_TM %
%   B26:25/0  GET_3_HT_PH_GAS_WRN %
% Rung: 2 %
% TITLE: HIGH TEMP GETTER PREHEATER %
SOR NEQ N10:0 N9:6 BST GEQ I:6.2 N7:19 NEQ I:6.2 N7:81 NXB GEQ I:6.1 N7:19 NEQ I:6.1 N7:81 BND XIC B26:10/2 BST MOV N18:22 T4:164.PRE NXB TON T4:164 1.0 5 0 NXB XIC T4:164/DN OTE B26:19/1 BND EOR
%   N10:0  SYSTEM_STATE  "STATE The current state of the system" %
%   N9:6  SYSTEM_PURGE %
%   I:6.2  GET_3_PH_OUTER_TC  "TC12" %
%   N7:19  GET_HT_PH_ALM_SP %
%   N7:81  TC_OPEN_SP  "CONFIG The value read by an open TC input" %
%   I:6.1  GET_3_PH_INNER_TC  "TC11" %
%   B26:10/2  GET_HT_PH_ALM_EN %
%   N18:22  GET_HT_PH_ALM_DLY %
%   T4:164  GET_3_HT_PH_ALM_TMR %
%   B26:19/1  GET_3_HT_PH_ALARM %

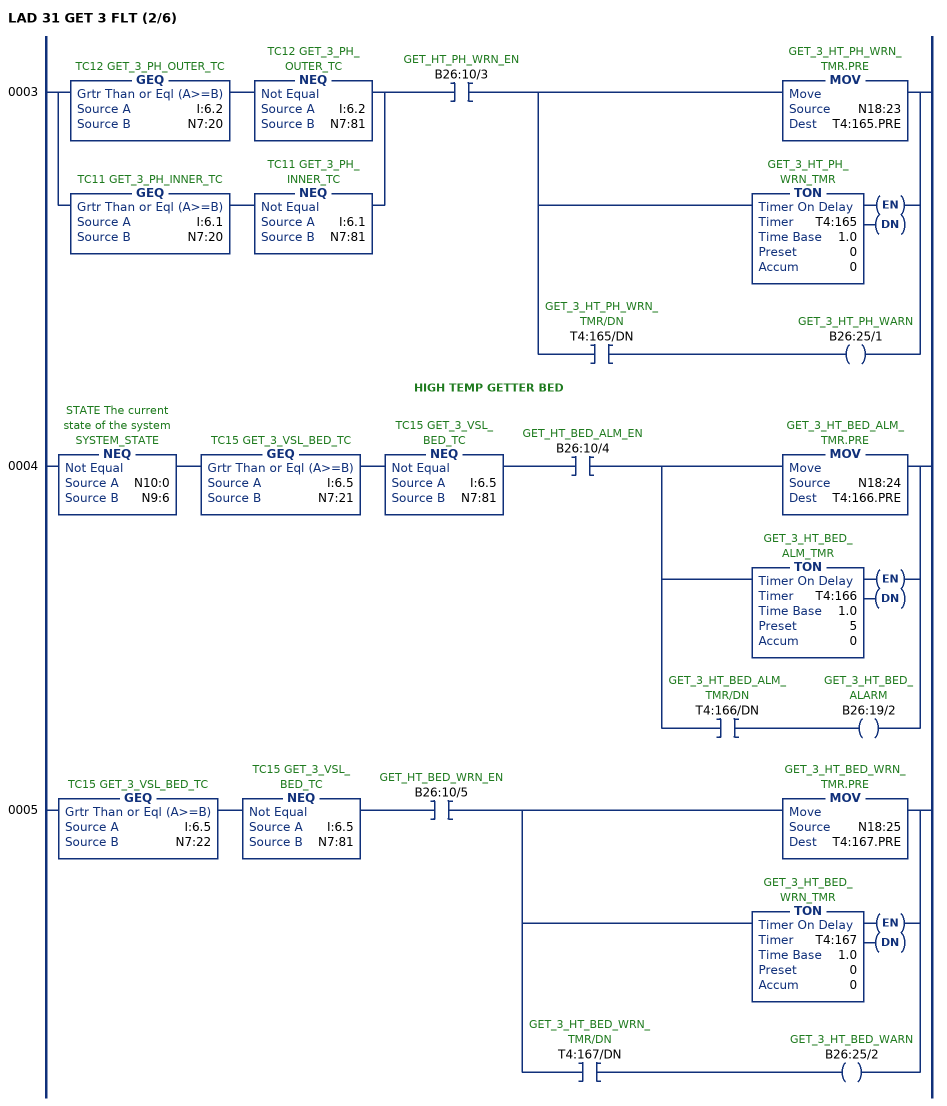
% Rung: 3 %
SOR BST GEQ I:6.2 N7:20 NEQ I:6.2 N7:81 NXB GEQ I:6.1 N7:20 NEQ I:6.1 N7:81 BND XIC B26:10/3 BST MOV N18:23 T4:165.PRE NXB TON T4:165 1.0 0 0 NXB XIC T4:165/DN OTE B26:25/1 BND EOR
%   I:6.2  GET_3_PH_OUTER_TC  "TC12" %
%   N7:20  GET_HT_PH_WRN_SP %
%   N7:81  TC_OPEN_SP  "CONFIG The value read by an open TC input" %
%   I:6.1  GET_3_PH_INNER_TC  "TC11" %
%   B26:10/3  GET_HT_PH_WRN_EN %
%   N18:23  GET_HT_PH_WRN_DLY %
%   T4:165  GET_3_HT_PH_WRN_TMR %
%   B26:25/1  GET_3_HT_PH_WARN %
% Rung: 4 %
% TITLE: HIGH TEMP GETTER BED %
SOR NEQ N10:0 N9:6 GEQ I:6.5 N7:21 NEQ I:6.5 N7:81 XIC B26:10/4 BST MOV N18:24 T4:166.PRE NXB TON T4:166 1.0 5 0 NXB XIC T4:166/DN OTE B26:19/2 BND EOR
%   N10:0  SYSTEM_STATE  "STATE The current state of the system" %
%   N9:6  SYSTEM_PURGE %
%   I:6.5  GET_3_VSL_BED_TC  "TC15" %
%   N7:21  GET_HT_BED_ALM_SP %
%   N7:81  TC_OPEN_SP  "CONFIG The value read by an open TC input" %
%   B26:10/4  GET_HT_BED_ALM_EN %
%   N18:24  GET_HT_BED_ALM_DLY %
%   T4:166  GET_3_HT_BED_ALM_TMR %
%   B26:19/2  GET_3_HT_BED_ALARM %
% Rung: 5 %
SOR GEQ I:6.5 N7:22 NEQ I:6.5 N7:81 XIC B26:10/5 BST MOV N18:25 T4:167.PRE NXB TON T4:167 1.0 0 0 NXB XIC T4:167/DN OTE B26:25/2 BND EOR
%   I:6.5  GET_3_VSL_BED_TC  "TC15" %
%   N7:22  GET_HT_BED_WRN_SP %
%   N7:81  TC_OPEN_SP  "CONFIG The value read by an open TC input" %
%   B26:10/5  GET_HT_BED_WRN_EN %
%   N18:25  GET_HT_BED_WRN_DLY %
%   T4:167  GET_3_HT_BED_WRN_TMR %
%   B26:25/2  GET_3_HT_BED_WARN %

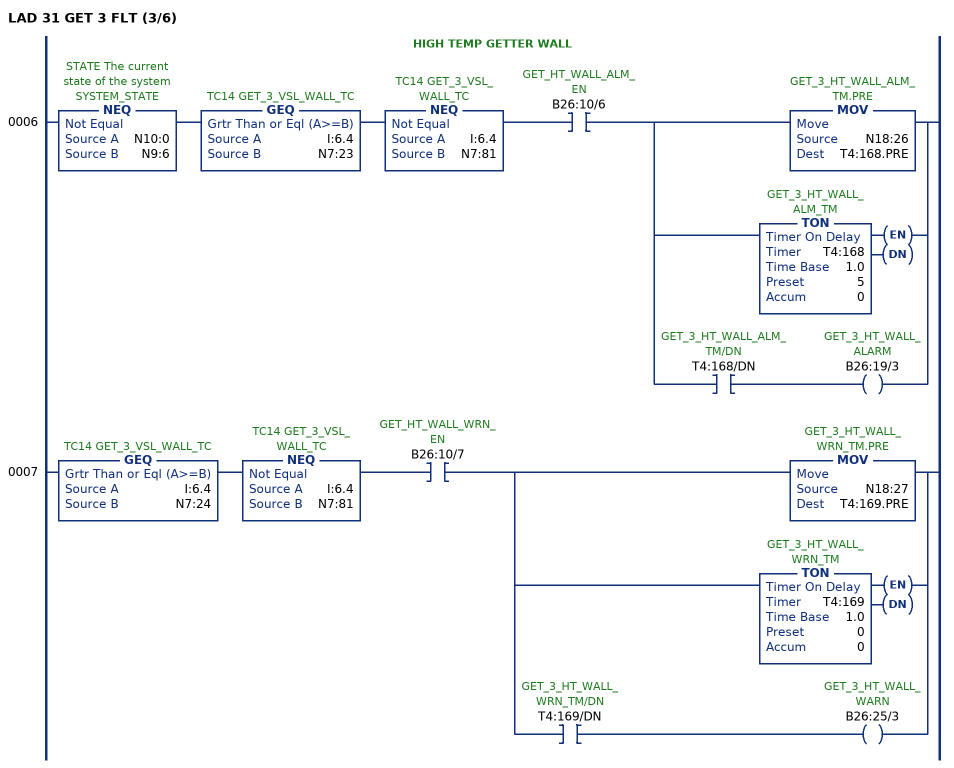
% Rung: 6 %
% TITLE: HIGH TEMP GETTER WALL %
SOR NEQ N10:0 N9:6 GEQ I:6.4 N7:23 NEQ I:6.4 N7:81 XIC B26:10/6 BST MOV N18:26 T4:168.PRE NXB TON T4:168 1.0 5 0 NXB XIC T4:168/DN OTE B26:19/3 BND EOR
%   N10:0  SYSTEM_STATE  "STATE The current state of the system" %
%   N9:6  SYSTEM_PURGE %
%   I:6.4  GET_3_VSL_WALL_TC  "TC14" %
%   N7:23  GET_HT_WALL_ALM_SP %
%   N7:81  TC_OPEN_SP  "CONFIG The value read by an open TC input" %
%   B26:10/6  GET_HT_WALL_ALM_EN %
%   N18:26  GET_HT_WALL_ALM_DLY %
%   T4:168  GET_3_HT_WALL_ALM_TM %
%   B26:19/3  GET_3_HT_WALL_ALARM %
% Rung: 7 %
SOR GEQ I:6.4 N7:24 NEQ I:6.4 N7:81 XIC B26:10/7 BST MOV N18:27 T4:169.PRE NXB TON T4:169 1.0 0 0 NXB XIC T4:169/DN OTE B26:25/3 BND EOR
%   I:6.4  GET_3_VSL_WALL_TC  "TC14" %
%   N7:24  GET_HT_WALL_WRN_SP %
%   N7:81  TC_OPEN_SP  "CONFIG The value read by an open TC input" %
%   B26:10/7  GET_HT_WALL_WRN_EN %
%   N18:27  GET_HT_WALL_WRN_DLY %
%   T4:169  GET_3_HT_WALL_WRN_TM %
%   B26:25/3  GET_3_HT_WALL_WARN %

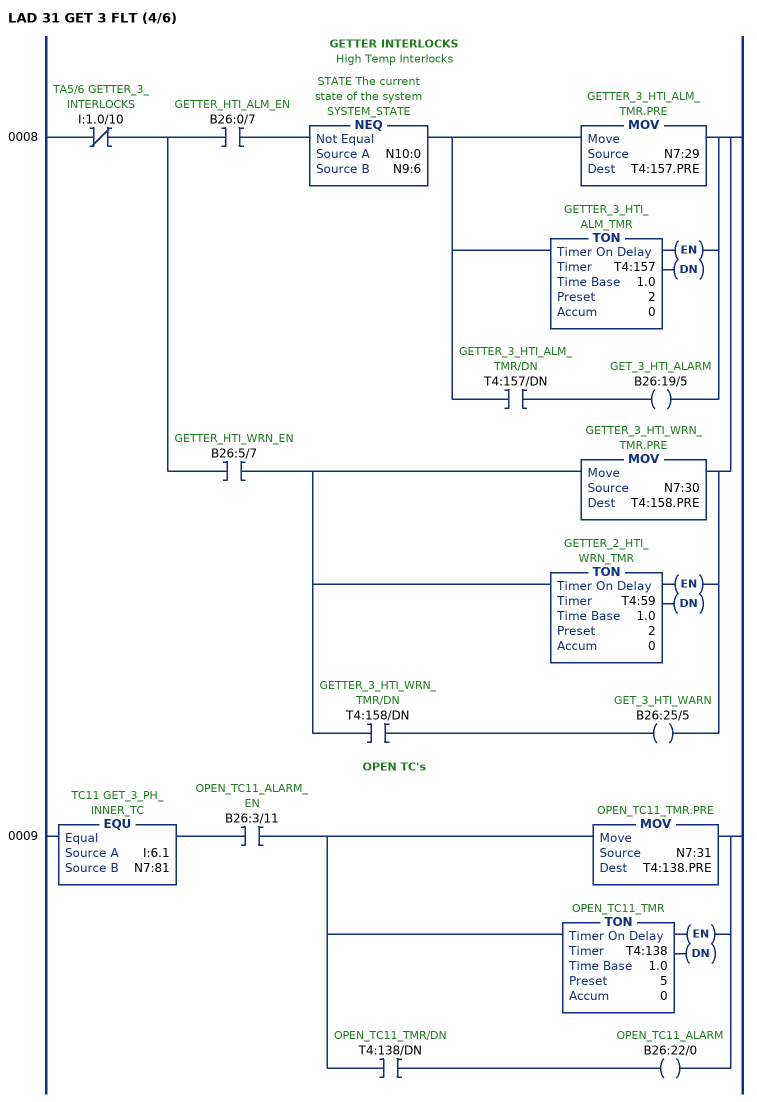
% Rung: 8 %
% TITLE: GETTER INTERLOCKS %
% High Temp Interlocks %
SOR XIO I:1.0/10 BST XIC B26:0/7 NEQ N10:0 N9:6 BST MOV N7:29 T4:157.PRE NXB TON T4:157 1.0 2 0 NXB XIC T4:157/DN OTE B26:19/5 BND NXB XIC B26:5/7 BST MOV N7:30 T4:158.PRE NXB TON T4:59 1.0 2 0 NXB XIC T4:158/DN OTE B26:25/5 BND BND EOR
%   I:1.0/10  GETTER_3_INTERLOCKS  "TA5/6" %
%   B26:0/7  GETTER_HTI_ALM_EN %
%   N10:0  SYSTEM_STATE  "STATE The current state of the system" %
%   N9:6  SYSTEM_PURGE %
%   N7:29  GETTER_HTI_ALM_DLY %
%   T4:157  GETTER_3_HTI_ALM_TMR %
%   B26:19/5  GET_3_HTI_ALARM %
%   B26:5/7  GETTER_HTI_WRN_EN %
%   N7:30  GETTER_HTI_WRN_DLY %
%   T4:158  GETTER_3_HTI_WRN_TMR %
%   T4:59  GETTER_2_HTI_WRN_TMR %
%   B26:25/5  GET_3_HTI_WARN %
% Rung: 9 %
% TITLE: OPEN TC's %
SOR EQU I:6.1 N7:81 XIC B26:3/11 BST MOV N7:31 T4:138.PRE NXB TON T4:138 1.0 5 0 NXB XIC T4:138/DN OTE B26:22/0 BND EOR
%   I:6.1  GET_3_PH_INNER_TC  "TC11" %
%   N7:81  TC_OPEN_SP  "CONFIG The value read by an open TC input" %
%   B26:3/11  OPEN_TC11_ALARM_EN %
%   N7:31  OPEN_TC_DLY %
%   T4:138  OPEN_TC11_TMR %
%   B26:22/0  OPEN_TC11_ALARM %

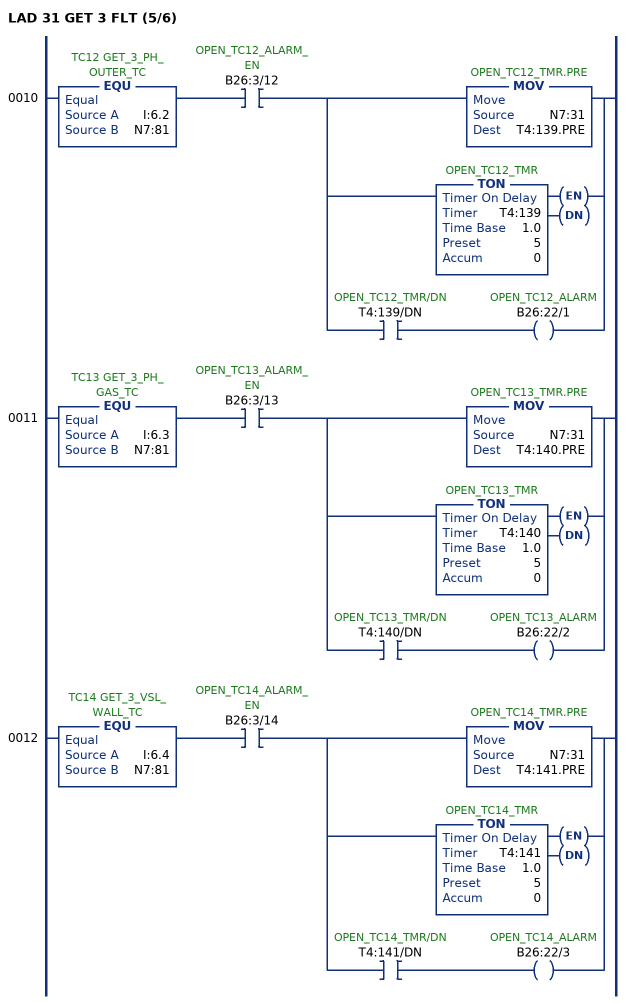
% Rung: 10 %
SOR EQU I:6.2 N7:81 XIC B26:3/12 BST MOV N7:31 T4:139.PRE NXB TON T4:139 1.0 5 0 NXB XIC T4:139/DN OTE B26:22/1 BND EOR
%   I:6.2  GET_3_PH_OUTER_TC  "TC12" %
%   N7:81  TC_OPEN_SP  "CONFIG The value read by an open TC input" %
%   B26:3/12  OPEN_TC12_ALARM_EN %
%   N7:31  OPEN_TC_DLY %
%   T4:139  OPEN_TC12_TMR %
%   B26:22/1  OPEN_TC12_ALARM %
% Rung: 11 %
SOR EQU I:6.3 N7:81 XIC B26:3/13 BST MOV N7:31 T4:140.PRE NXB TON T4:140 1.0 5 0 NXB XIC T4:140/DN OTE B26:22/2 BND EOR
%   I:6.3  GET_3_PH_GAS_TC  "TC13" %
%   N7:81  TC_OPEN_SP  "CONFIG The value read by an open TC input" %
%   B26:3/13  OPEN_TC13_ALARM_EN %
%   N7:31  OPEN_TC_DLY %
%   T4:140  OPEN_TC13_TMR %
%   B26:22/2  OPEN_TC13_ALARM %
% Rung: 12 %
SOR EQU I:6.4 N7:81 XIC B26:3/14 BST MOV N7:31 T4:141.PRE NXB TON T4:141 1.0 5 0 NXB XIC T4:141/DN OTE B26:22/3 BND EOR
%   I:6.4  GET_3_VSL_WALL_TC  "TC14" %
%   N7:81  TC_OPEN_SP  "CONFIG The value read by an open TC input" %
%   B26:3/14  OPEN_TC14_ALARM_EN %
%   N7:31  OPEN_TC_DLY %
%   T4:141  OPEN_TC14_TMR %
%   B26:22/3  OPEN_TC14_ALARM %

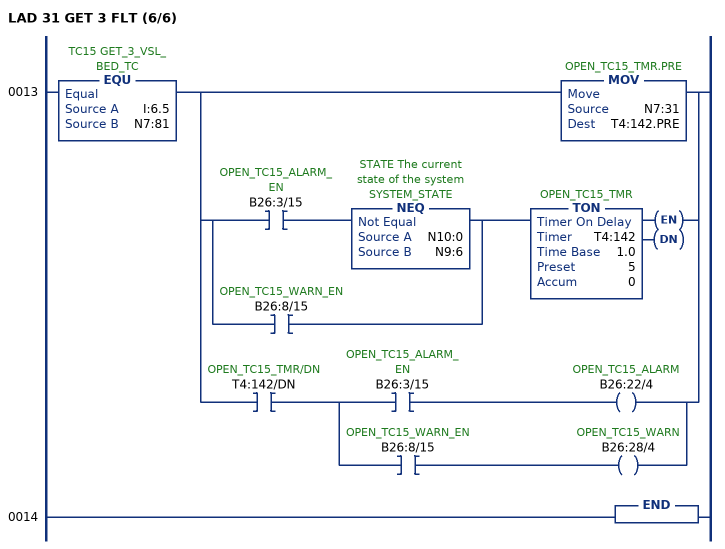
% Rung: 13 %
SOR EQU I:6.5 N7:81 BST MOV N7:31 T4:142.PRE NXB BST XIC B26:3/15 NEQ N10:0 N9:6 NXB XIC B26:8/15 BND TON T4:142 1.0 5 0 NXB XIC T4:142/DN BST XIC B26:3/15 OTE B26:22/4 NXB XIC B26:8/15 OTE B26:28/4 BND BND EOR
%   I:6.5  GET_3_VSL_BED_TC  "TC15" %
%   N7:81  TC_OPEN_SP  "CONFIG The value read by an open TC input" %
%   N7:31  OPEN_TC_DLY %
%   T4:142  OPEN_TC15_TMR %
%   B26:3/15  OPEN_TC15_ALARM_EN %
%   N10:0  SYSTEM_STATE  "STATE The current state of the system" %
%   N9:6  SYSTEM_PURGE %
%   B26:8/15  OPEN_TC15_WARN_EN %
%   B26:22/4  OPEN_TC15_ALARM %
%   B26:28/4  OPEN_TC15_WARN %
% Rung: 14 %
SOR END EOR

LADDER 32 "GET 3"
